{attribute 'linkalways'} 
{attribute 'no_explicit_call' := 'This FB is a CLASS and must be accessed using methods or properties'}
{attribute 'enable_dynamic_creation'}
FUNCTION_BLOCK DictionaryTreeNode EXTENDS Disposable IMPLEMENTS I_DictionaryTreeNode
VAR
	_key : T_MAXSTRING;
	pBuffer : POINTER TO BYTE;
	bufferSize : UDINT;
    _height : DINT;
    _left : I_DictionaryTreeNode;
    _right : I_DictionaryTreeNode;
END_VAR

METHOD PUBLIC Clone
VAR_INPUT
	Node : I_DictionaryTreeNode;
END_VAR
DestroyBuffer();
CreateBuffer(Node.NodeBufferSize);
CopySourceToBuffer(Node.NodeBufferPointer);
_key := Node.Key;
END_METHOD

METHOD PRIVATE CopyBufferToDestination
VAR_INPUT
	DestinationAddress : PVOID;
END_VAR
MEMCPY(DestinationAddress, pBuffer, bufferSize);
END_METHOD

METHOD PRIVATE CopySourceToBuffer
VAR_INPUT
	SourceAddress : PVOID;
END_VAR
MEMCPY(pBuffer, SourceAddress, bufferSize);
END_METHOD

METHOD PRIVATE CreateBuffer
VAR_INPUT
	SizeInBytes : UDINT;
END_VAR
bufferSize := SizeInBytes;
pBuffer := __NEW(BYTE, SizeInBytes);
END_METHOD

PROPERTY PUBLIC DataSize : UDINT
GET
DataSize := bufferSize;
END_GET
END_PROPERTY

METHOD PRIVATE DestroyBuffer
VAR_INPUT
END_VAR
IF pBuffer = 0 THEN
	RETURN;
END_IF

__DELETE(pBuffer);
bufferSize := 0;
END_METHOD

METHOD PUBLIC Equals : BOOL
VAR_INPUT
	Symbol : ANY;
END_VAR
IF pBuffer = 0 THEN
	RETURN;
END_IF

IF bufferSize <> DINT_TO_UDINT(symbol.diSize) THEN
	RETURN;
END_IF

Equals := MEMCMP(Symbol.pValue, pBuffer, bufferSize) = 0;
END_METHOD

METHOD FB_exit : BOOL
VAR_INPUT
	bInCopyCode : BOOL; // if TRUE, the exit method is called for exiting an instance that is copied afterwards (online change).
END_VAR
IF bInCopyCode THEN
	RETURN;
END_IF

DestroyBuffer();
END_METHOD

METHOD FB_init : BOOL
VAR_INPUT
	bInitRetains : BOOL; // if TRUE, the retain variables are initialized (warm start / cold start)
	bInCopyCode : BOOL;  // if TRUE, the instance afterwards gets moved into the copy code (online change)
	NodeKey : T_MAXSTRING;
	NodeSource : ANY;
END_VAR
_key := NodeKey;
CreateBuffer(DINT_TO_UDINT(NodeSource.diSize));
CopySourceToBuffer(NodeSource.pValue);
END_METHOD

PROPERTY PUBLIC Height : DINT
GET
Height := _height;
END_GET
SET // PUBLIC
_height := Height;
END_SET
END_PROPERTY

PROPERTY PUBLIC Key : T_MAXSTRING
GET
Key := _key;
END_GET
END_PROPERTY

PROPERTY PUBLIC Left : I_DictionaryTreeNode
GET
Left := _left;
END_GET
SET
_left := Left;
END_SET
END_PROPERTY

PROPERTY PUBLIC NodeBufferPointer : Pointer To Byte
GET
NodeBufferPointer := pBuffer;
END_GET
END_PROPERTY

PROPERTY PUBLIC NodeBufferSize : UDINT
GET
NodeBufferSize := bufferSize;
END_GET
END_PROPERTY

METHOD Reinitialize
VAR_INPUT
	Key : T_MAXSTRING;
	Source : ANY;
END_VAR
_key := Key;

IF pBuffer <> 0 THEN
	DestroyBuffer();
END_IF

CreateBuffer(DINT_TO_UDINT(Source.diSize));
CopySourceToBuffer(Source.pValue);
END_METHOD

PROPERTY PUBLIC Right : I_DictionaryTreeNode
GET
Right := _right;
END_GET
SET
_right := Right;
END_SET
END_PROPERTY

METHOD TryGet : BOOL
VAR_INPUT
	Destination	: ANY;
END_VAR
TryGet := TryGetTo(Destination.pValue, DINT_TO_UDINT(Destination.diSize));
END_METHOD

METHOD TryGetTo : BOOL
VAR_INPUT
	DestinationAddress : PVOID;
	DestinationSize : UDINT;
END_VAR
IF pBuffer = 0 THEN
	RETURN;
END_IF

IF bufferSize <> DestinationSize THEN
	RETURN;
END_IF

CopyBufferToDestination(DestinationAddress);
TryGetTo := TRUE;
END_METHOD

END_FUNCTION_BLOCK

(* stored: Version 1.1.0.1, ProductVersion 3.1.4024.12
   POU DictionaryTreeNode: Id {4678eec6-e97b-0636-2914-7ff5f441eaef}, SpecialFunc None
   Folder Constructor: Id {0f890dd3-beaf-007b-0699-78b1ea3f6ba9}
   Folder Destructor: Id {fd7f6b61-274d-0c38-03cb-112a20bea0ef}
   Folder Private: Id {9e8fa089-e3cf-0b45-2628-c6e744d7beeb}
   Method Clone: Id {22a9bda3-ae13-0e42-0e32-3cb9d3361f3b}
   Method CopyBufferToDestination: Id {c38d820e-319f-02cb-2abb-e2d6a9beb266}
   Method CopySourceToBuffer: Id {91cf1b29-0557-0488-1ee8-d6eda2f40862}
   Method CreateBuffer: Id {8790e7f8-b4eb-01d6-3738-05211e965826}
   Property DataSize: Id {6303471a-7abf-0951-0f3c-aa0e62ce08ae}
   Get Get: Id {5da9af5a-4b3f-098b-3082-6037532192e4}
   Method DestroyBuffer: Id {cec4953f-c967-04cc-3b01-0e4ed4fb6ee8}
   Method Equals: Id {50c9dac2-3c86-0a26-2040-adb9fce9caf9}
   Method FB_exit: Id {acb933af-0ccf-0313-3019-626ed07bb00e}
   Method FB_init: Id {d3a86937-eb89-05a7-0d7c-647e8efcb5e6}
   Property Height: Id {701257fd-4916-062b-06a1-3d0e71924719}
   Get Get: Id {6fcafdd8-ae6f-0194-30a9-e36c50224e8d}
   Set Set: Id {21cea8e7-254b-06b4-110e-5a4d03ac7bef}
   Property Key: Id {28bd6992-4b51-03dd-3c99-7cd6a754cf70}
   Get Get: Id {7a83318d-a2a0-0cda-3190-ac1be70fca6a}
   Property Left: Id {da7e8da7-b52f-0597-0b0f-bad04ffeef78}
   Get Get: Id {677e498e-fd77-0bc2-2d72-df4e8bc110a3}
   Set Set: Id {bb3e3275-4339-09c8-296a-e696649f35e0}
   Property NodeBufferPointer: Id {b1fad07b-2b15-0eeb-2fb0-b02abb1acbe2}
   Get Get: Id {fca05c78-c992-0ea7-28b3-e2ec06dc11ce}
   Property NodeBufferSize: Id {60bc77e9-12cb-0d23-228d-1b2b3aebe161}
   Get Get: Id {7678eb28-3424-0be4-3a28-7b2d8fe8b4b0}
   Method Reinitialize: Id {5464e52b-aadd-0892-250a-ef554f7a16aa}
   Property Right: Id {b07d37d0-e2ed-055d-2a11-681a1d4a1e4f}
   Get Get: Id {540edd64-22e3-032f-0945-319afe7962f6}
   Set Set: Id {52e1865b-6bf0-070d-0996-dfd5a5e038c2}
   Method TryGet: Id {2990a6b5-b0f5-09bb-3d58-0785c0efd4c6}
   Method TryGetTo: Id {f23ae461-6805-07a8-04d0-28363c28779d} *)
